// TIA Portal project "Project9" (V15.1)
// motor yıldız ücgen

(* hardware
DEVICE "S7-1200 station_1"  S7-1200 Station
   slot 0: "Rack_0"  S7-1200 Rack  Rack  V1.0
   slot 1: "PLC_1"  CPU 1214C AC/DC/Rly  6ES7 214-1BG40-0XB0  V4.2
*)

// ===== PLC "PLC_1"  CPU 1214C AC/DC/Rly =====

VAR_GLOBAL   // PLC tag table "Default tag table"
   "start" AT %I0.0 : Bool;
   "stop" AT %I0.1 : Bool;
   "ana kont" AT %Q0.2 : Bool;
   "ucgen" AT %Q0.3 : Bool;
   "yıldız" AT %Q0.4 : Bool;
END_VAR

// folder: System blocks/Program resources

DATA_BLOCK "timer1"   // DB1
{ S7_Optimized_Access := 'TRUE' }
AUTHOR : Simatic
FAMILY : IEC
NAME : IEC_TMR
VERSION : 1.0
// stored: InstanceOfName IEC_TIMER
"IEC_TIMER"
BEGIN
END_DATA_BLOCK

// folder: (top level)

ORGANIZATION_BLOCK "Main"   // OB1, LAD, ProgramCycle
TITLE = "Main Program Sweep (Cycle)"
{ S7_Optimized_Access := 'TRUE' }
VERSION : 0.1
   VAR_INPUT
      Initial_Call : Bool;   // Initial call of this OB
      Remanence : Bool;   // =True, if remanent data are available
   END_VAR
BEGIN

REGION Network 1
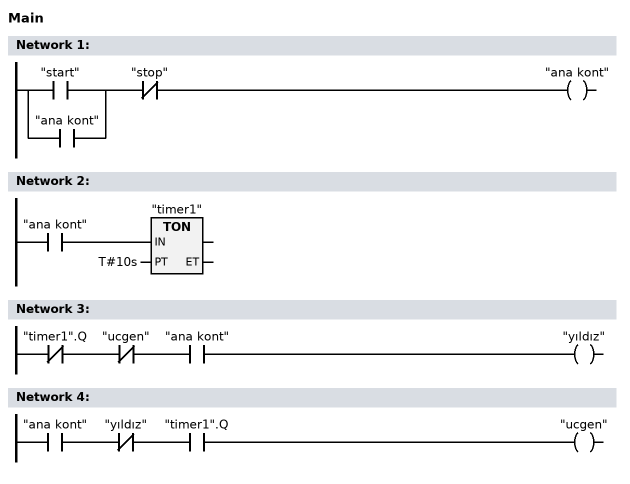
   RUNG wire#powerrail
      Contact( "start" )
      wire#w1
      I_Contact( "stop" )
      Coil( "ana kont" )
   END_RUNG
   RUNG wire#powerrail
      Contact( "ana kont" )
   END_RUNG wire#w1
   // the same network as SCL:
   "ana kont" := ("start" OR "ana kont") AND NOT "stop";
END_REGION

REGION Network 2
   "timer1".TON(IN := "ana kont", PT := T#10s);
END_REGION

REGION Network 3
   RUNG wire#powerrail
      I_Contact( "timer1".Q )
      I_Contact( "ucgen" )
      Contact( "ana kont" )
      Coil( "yıldız" )
   END_RUNG
   // the same network as SCL:
   "yıldız" := NOT "timer1".Q AND NOT "ucgen" AND "ana kont";
END_REGION

REGION Network 4
   RUNG wire#powerrail
      Contact( "ana kont" )
      I_Contact( "yıldız" )
      Contact( "timer1".Q )
      Coil( "ucgen" )
   END_RUNG
   // the same network as SCL:
   "ucgen" := "ana kont" AND NOT "yıldız" AND "timer1".Q;
END_REGION
END_ORGANIZATION_BLOCK